// TIA Portal project "Project" (V15)

(* hardware
DEVICE "S7-1200 station_1"  S7-1200 Station
   slot 0: "Rack_0"  S7-1200 Rack  Rack  V1.0
   slot 1: "PLC_1"  CPU 1214C DC/DC/DC  6ES7 214-1AG40-0XB0  V4.2
DEVICE "HMI_1"  TP1200 Comfort
   slot 0: "HMI_1"  TP1200 Comfort  6AV2 124-0MC01-0AX0  15.0.0.0
   slot 1: "HMI_RT_1"  TP1200 Comfort  6AV2 124-0MC01-0AX0  15.0.0.0
   slot 5: "HMI_1.IE_CP_1"  PROFINET Interface  15.0.0.0
      slot 1: "PROFINET Interface_1"  PROFINET Interface
         slot 1: "Port_1"  Port
         slot 2: "Port_2"  Port
   slot 7: "HMI_1.MPI/DP_CP_1"  MPI/DP Interface  15.0.0.0
*)

// ===== PLC "PLC_1"  CPU 1214C DC/DC/DC =====

VAR_GLOBAL   // PLC tag table "Default tag table"
   "Start" AT %M0.0 : Bool;
   "Stop" AT %M0.1 : Bool;
   "Run" AT %M0.2 : Bool;
   "Low" AT %M0.3 : Bool;
   "Reset" AT %M0.4 : Bool;
   "Sensor_Low" AT %M0.5 : Bool;
   "Piston_Low" AT %Q0.0 : Bool;
   "High" AT %M0.6 : Bool;
   "Sensor_High" AT %M0.7 : Bool;
   "Piston_High" AT %Q0.1 : Bool;
   "Medium" AT %M1.0 : Bool;
   "Sensor_Medium" AT %M1.1 : Bool;
   "Piston_Medium" AT %Q0.2 : Bool;
END_VAR

DATA_BLOCK "Control_Piston_Low_DB"   // DB1
{ S7_Optimized_Access := 'TRUE' }
VERSION : 0.1
// stored: InstanceOfName Control_Piston
"Control_Piston"
BEGIN
END_DATA_BLOCK

DATA_BLOCK "Control_Piston_High_DB"   // DB2
{ S7_Optimized_Access := 'TRUE' }
VERSION : 0.1
// stored: InstanceOfName Control_Piston
"Control_Piston"
BEGIN
END_DATA_BLOCK

DATA_BLOCK "Control_Piston_Med_DB"   // DB3
{ S7_Optimized_Access := 'TRUE' }
VERSION : 0.1
// stored: InstanceOfName Control_Piston
"Control_Piston"
BEGIN
END_DATA_BLOCK

DATA_BLOCK "DB_Main"   // DB4
{ S7_Optimized_Access := 'TRUE' }
VERSION : 0.1
   VAR
      Pos_edge_1 : Bool;
      Pos_edge_2 : Bool;
      Pos_edge_3 : Bool;
      Number_of_low_boxes : Int;
      Number_of_med_boxes : Int;
      Number_of_high_boxes : Int;
   END_VAR
BEGIN
END_DATA_BLOCK

// folder: System blocks/Program resources

DATA_BLOCK "IEC_Counter_0_DB"   // DB5
{ S7_Optimized_Access := 'TRUE' }
AUTHOR : Simatic
FAMILY : IEC
NAME : CNTR
VERSION : 1.0
// stored: InstanceOfName IEC_COUNTER
"IEC_COUNTER"
BEGIN
END_DATA_BLOCK

DATA_BLOCK "IEC_Counter_1_DB"   // DB6
{ S7_Optimized_Access := 'TRUE' }
AUTHOR : Simatic
FAMILY : IEC
NAME : CNTR
VERSION : 1.0
// stored: InstanceOfName IEC_COUNTER
"IEC_COUNTER"
BEGIN
END_DATA_BLOCK

DATA_BLOCK "IEC_Counter_2_DB"   // DB7
{ S7_Optimized_Access := 'TRUE' }
AUTHOR : Simatic
FAMILY : IEC
NAME : CNTR
VERSION : 1.0
// stored: InstanceOfName IEC_COUNTER
"IEC_COUNTER"
BEGIN
END_DATA_BLOCK

// folder: (top level)

FUNCTION_BLOCK "Single_box_behaviour"   // FB1, LAD
{ S7_Optimized_Access := 'TRUE' }
VERSION : 0.1
// Khối quản lý hành vi của từng hộp
   VAR_INPUT
      Low_box_in : Bool;
      Start : Bool;
      Stop : Bool;
      Run : Bool;
      Reset : Bool;
      Maximum_time : Time;
      Maximum_time_int : Int;
   END_VAR
   VAR_OUTPUT
      Current_time : Int;
      Animation_run_out : Bool;
   END_VAR
   VAR
      Animation_run : Bool;
      IEC_Timer_0_Instance : TON_TIME;
      Low__timer_acc : Time;
      Current_time_mem : Int;
      Halting : Bool;
      Pos_edge_1 : Bool;
   END_VAR
   VAR_TEMP
      Low__timer_acc_int : Int;
   END_VAR
   VAR_TEMP   // added for the SCL form of the ladder/FBD networks
      _w1 : Bool;
   END_VAR
BEGIN

REGION Network 1
   // Cho animation chạy khi có tín hiệu xung cạnh lên hoặc tiếp tục khi đang stop
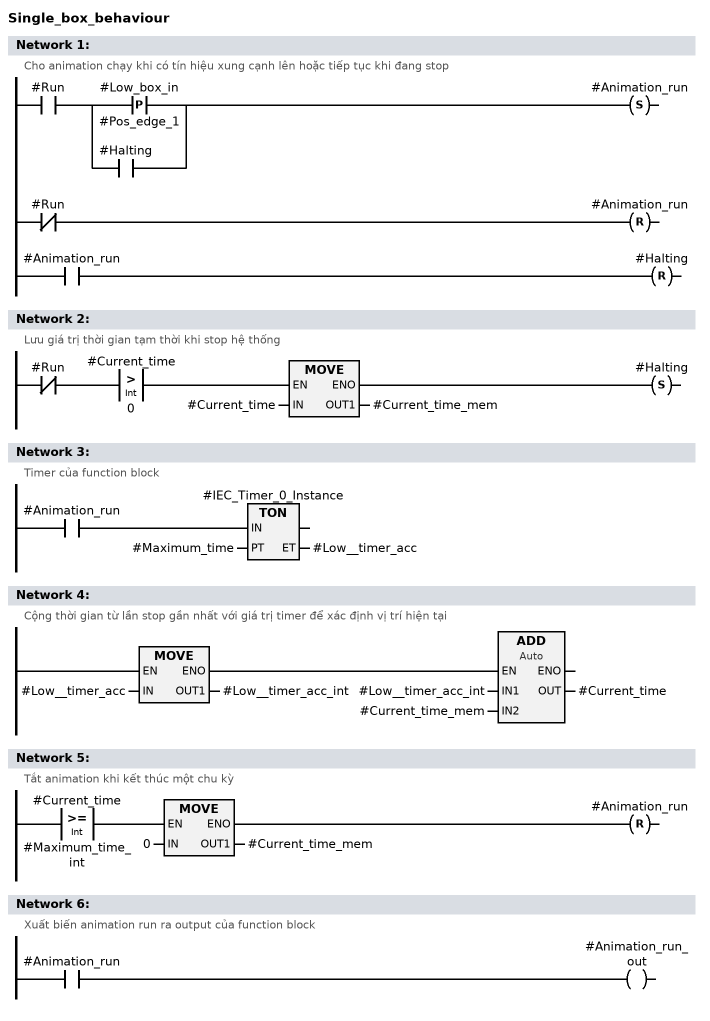
   RUNG wire#powerrail
      Contact( #Run )
      wire#w1
      P_Contact(operand := #Low_box_in, bit := #Pos_edge_1)
      wire#w2
      S_Coil( #Animation_run )
   END_RUNG
   RUNG wire#w1
      Contact( #Halting )
   END_RUNG wire#w2
   RUNG wire#powerrail
      I_Contact( #Run )
      R_Coil( #Animation_run )
   END_RUNG
   RUNG wire#powerrail
      Contact( #Animation_run )
      R_Coil( #Halting )
   END_RUNG
   // the same network as SCL:
   #_w1 := #Run AND #Low_box_in AND NOT #Pos_edge_1;   // rising edge of #Low_box_in
   #Pos_edge_1 := #Low_box_in;
   IF #_w1 OR (#Run AND #Halting) THEN #Animation_run := TRUE; END_IF;
   IF NOT #Run THEN #Animation_run := FALSE; END_IF;
   IF #Animation_run THEN #Halting := FALSE; END_IF;
END_REGION

REGION Network 2
   // Lưu giá trị thời gian tạm thời khi stop hệ thống
   RUNG wire#powerrail
      I_Contact( #Run )
      { S7_Templates := "SrcType := Int" } GT_Contact(in1 := #Current_time, in2 := 0)
      Move(in := #Current_time, out1 => #Current_time_mem)
      S_Coil( #Halting )
   END_RUNG
   // the same network as SCL:
   IF NOT #Run AND (#Current_time > 0) THEN
       #Current_time_mem := #Current_time;
       #Halting := TRUE;
   END_IF;
END_REGION

REGION Network 3
   // Timer của function block
   #IEC_Timer_0_Instance(IN := #Animation_run, PT := #Maximum_time, ET => #Low__timer_acc);   // TON
END_REGION

REGION Network 4
   // Cộng thời gian từ lần stop gần nhất với giá trị timer để xác định vị trí hiện tại
   RUNG wire#powerrail
      Move(in := #Low__timer_acc, out1 => #Low__timer_acc_int)
      Add(in1 := #Low__timer_acc_int, in2 := #Current_time_mem, out => #Current_time)
   END_RUNG
   // the same network as SCL:
   #Low__timer_acc_int := #Low__timer_acc;
   #Current_time := #Low__timer_acc_int + #Current_time_mem;
END_REGION

REGION Network 5
   // Tắt animation khi kết thúc một chu kỳ
   RUNG wire#powerrail
      { S7_Templates := "SrcType := Int" } GE_Contact(in1 := #Current_time, in2 := #Maximum_time_int)
      Move(in := 0, out1 => #Current_time_mem)
      R_Coil( #Animation_run )
   END_RUNG
   // the same network as SCL:
   IF #Current_time >= #Maximum_time_int THEN
       #Current_time_mem := 0;
       #Animation_run := FALSE;
   END_IF;
END_REGION

REGION Network 6
   // Xuất biến animation run ra output của function block
   RUNG wire#powerrail
      Contact( #Animation_run )
      Coil( #Animation_run_out )
   END_RUNG
   // the same network as SCL:
   #Animation_run_out := #Animation_run;
END_REGION
END_FUNCTION_BLOCK

FUNCTION_BLOCK "Multiple_boxes_behaviour"   // FB2, LAD
{ S7_Optimized_Access := 'TRUE' }
VERSION : 0.1
// Khối quản lý hành vi của từng nhóm hộp (thấp, trung bình, cao)
   VAR_INPUT
      Low_box_in : Bool;
      Start : Bool;
      Stop : Bool;
      Run : Bool;
      Reset : Bool;
      Maximum_time : Time;
      Maximum_time_int : Int;
      Sensor_Activate_Time : Int;
      Sensor_Deactivate_Time : Int;
   END_VAR
   VAR_OUTPUT
      Sensor : Bool;
   END_VAR
   VAR
      Neg_edge_1 : Bool;
   END_VAR
   VAR RETAIN
      IEC_Counter_0_Instance : CTUD_INT;
   END_VAR
   VAR
      Animation_1 : Bool;
      Number_of_running_graphic : Int;
      Animation_2 : Bool;
      Current_Time_1 : Int;
      Current_Time_2 : Int;
      Animation_3 : Bool;
      Load_value : Int;
      Current_Time_3 : Int;
      Count_down : Bool;
      Neg_edge_2 : Bool;
      Neg_edge_3 : Bool;
      Number_of_boxes_on_conveyor_belt : Int;
      Single_box_animation_1 : Bool;
      Single_box_animation_2 : Bool;
      Single_box_animation_3 : Bool;
      Neg_edge_4 : Bool;
      Neg_edge_5 : Bool;
      Neg_edge_6 : Bool;
      Reset_counter : Bool;
      Animation_wait : Bool;
      Pos_edge_1 : Bool;
      Single_box_animation_4 : Bool;
      Current_Time_4 : Int;
      Animation_4 : Bool;
      Neg_edge_7 : Bool;
      Single_box_animation_5 : Bool;
      Current_Time_5 : Int;
      Animation_5 : Bool;
      Neg_edge_8 : Bool;
      Neg_edge_9 : Bool;
      Neg_edge_10 : Bool;
      IEC_Timer_0_Instance : TON_TIME;
      Single_box_animation_Instance_1 : "Single_box_behaviour";
      Single_box_animation_Instance_2 : "Single_box_behaviour";
      Single_box_animation_Instance_3 : "Single_box_behaviour";
      Single_box_animation_Instance_5 : "Single_box_behaviour";
      Single_box_animation_Instance_4 : "Single_box_behaviour";
   END_VAR
   VAR_TEMP
      temp_1 : Int;
   END_VAR
   VAR_TEMP   // added for the SCL form of the ladder/FBD networks
      _w1 : Bool;
   END_VAR
BEGIN

REGION Network 1
   // Reset các animation khi có tín hiệu reset
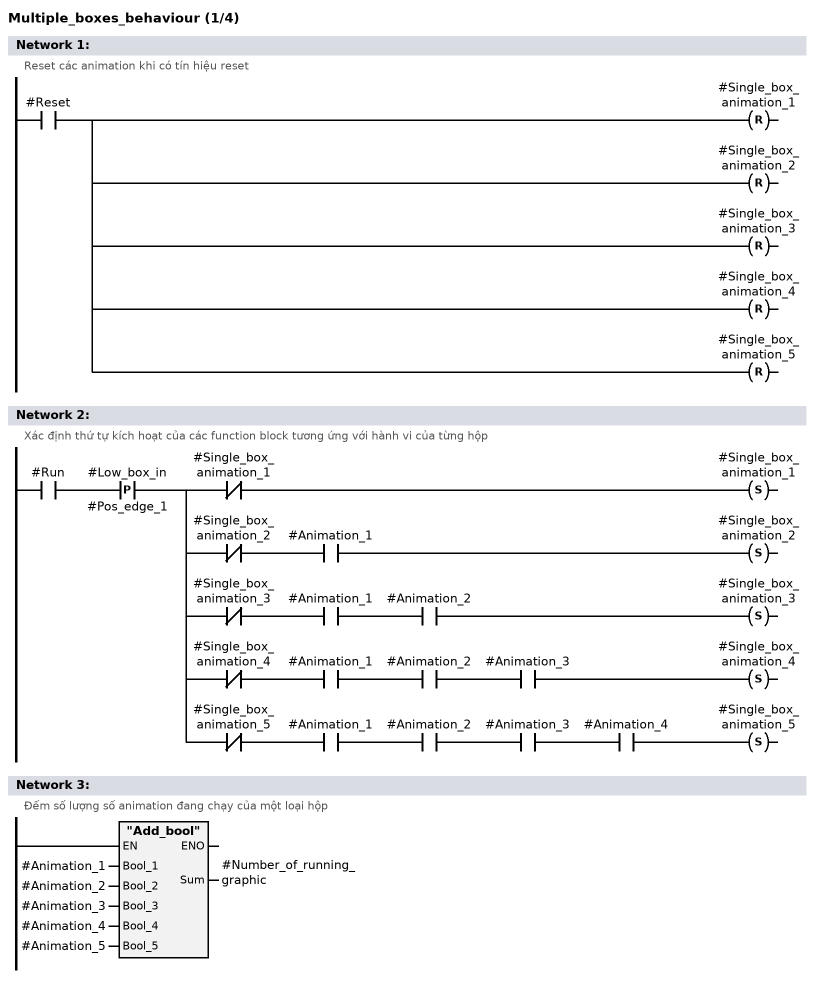
   RUNG wire#powerrail
      Contact( #Reset )
      wire#w1
      R_Coil( #Single_box_animation_1 )
   END_RUNG
   RUNG wire#w1
      R_Coil( #Single_box_animation_2 )
   END_RUNG
   RUNG wire#w1
      R_Coil( #Single_box_animation_3 )
   END_RUNG
   RUNG wire#w1
      R_Coil( #Single_box_animation_4 )
   END_RUNG
   RUNG wire#w1
      R_Coil( #Single_box_animation_5 )
   END_RUNG
   // the same network as SCL:
   IF #Reset THEN
       #Single_box_animation_1 := FALSE;
       #Single_box_animation_2 := FALSE;
       #Single_box_animation_3 := FALSE;
       #Single_box_animation_4 := FALSE;
       #Single_box_animation_5 := FALSE;
   END_IF;
END_REGION

REGION Network 2
   // Xác định thứ tự kích hoạt của các function block tương ứng với hành vi của từng hộp
   RUNG wire#powerrail
      Contact( #Run )
      P_Contact(operand := #Low_box_in, bit := #Pos_edge_1)
      wire#w1
      I_Contact( #Single_box_animation_1 )
      S_Coil( #Single_box_animation_1 )
   END_RUNG
   RUNG wire#w1
      I_Contact( #Single_box_animation_2 )
      Contact( #Animation_1 )
      S_Coil( #Single_box_animation_2 )
   END_RUNG
   RUNG wire#w1
      I_Contact( #Single_box_animation_3 )
      Contact( #Animation_1 )
      Contact( #Animation_2 )
      S_Coil( #Single_box_animation_3 )
   END_RUNG
   RUNG wire#w1
      I_Contact( #Single_box_animation_4 )
      Contact( #Animation_1 )
      Contact( #Animation_2 )
      Contact( #Animation_3 )
      S_Coil( #Single_box_animation_4 )
   END_RUNG
   RUNG wire#w1
      I_Contact( #Single_box_animation_5 )
      Contact( #Animation_1 )
      Contact( #Animation_2 )
      Contact( #Animation_3 )
      Contact( #Animation_4 )
      S_Coil( #Single_box_animation_5 )
   END_RUNG
   // the same network as SCL:
   #_w1 := #Run AND #Low_box_in AND NOT #Pos_edge_1;   // rising edge of #Low_box_in
   #Pos_edge_1 := #Low_box_in;
   IF #_w1 AND NOT #Single_box_animation_1 THEN #Single_box_animation_1 := TRUE; END_IF;
   IF #_w1 AND NOT #Single_box_animation_2 AND #Animation_1 THEN #Single_box_animation_2 := TRUE; END_IF;
   IF #_w1 AND NOT #Single_box_animation_3 AND #Animation_1 AND #Animation_2 THEN
       #Single_box_animation_3 := TRUE;
   END_IF;
   IF #_w1 AND NOT #Single_box_animation_4 AND #Animation_1 AND #Animation_2 AND #Animation_3 THEN
       #Single_box_animation_4 := TRUE;
   END_IF;
   IF #_w1 AND NOT #Single_box_animation_5 AND #Animation_1 AND #Animation_2 AND #Animation_3 AND #Animation_4 THEN
       #Single_box_animation_5 := TRUE;
   END_IF;
END_REGION

REGION Network 3
   // Đếm số lượng số animation đang chạy của một loại hộp
   RUNG wire#powerrail
      "Add_bool"(Bool_1 := #Animation_1, Bool_2 := #Animation_2, Bool_3 := #Animation_3, Bool_4 := #Animation_4, Bool_5 := #Animation_5, Sum => #Number_of_running_graphic)
   END_RUNG
   // the same network as SCL:
   "Add_bool"(Bool_1 := #Animation_1,
              Bool_2 := #Animation_2,
              Bool_3 := #Animation_3,
              Bool_4 := #Animation_4,
              Bool_5 := #Animation_5,
              Sum => #Number_of_running_graphic);
END_REGION

REGION Network 4
   // Function block xác định hành vi của hộp thứ 1
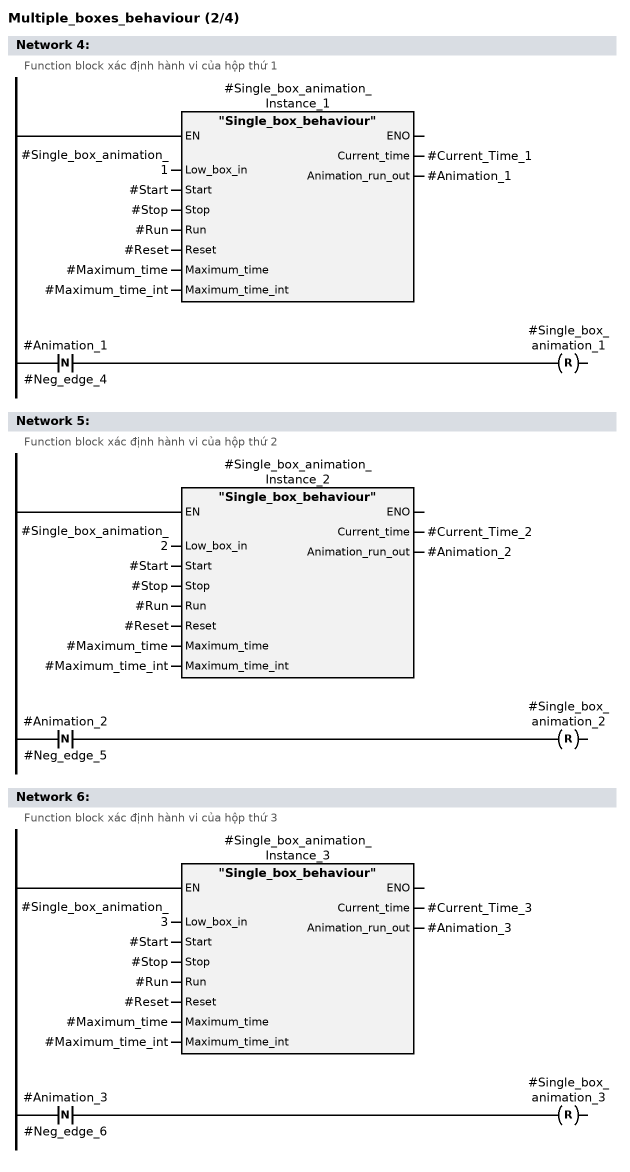
   RUNG wire#powerrail
      #Single_box_animation_Instance_1(Low_box_in := #Single_box_animation_1, Start := #Start, Stop := #Stop, Run := #Run, Reset := #Reset, Maximum_time := #Maximum_time, Maximum_time_int := #Maximum_time_int, Current_time => #Current_Time_1, Animation_run_out => #Animation_1)
   END_RUNG
   RUNG wire#powerrail
      N_Contact(operand := #Animation_1, bit := #Neg_edge_4)
      R_Coil( #Single_box_animation_1 )
   END_RUNG
   // the same network as SCL:
   #Single_box_animation_Instance_1(Low_box_in := #Single_box_animation_1,   // "Single_box_behaviour"
                           Start := #Start,
                           Stop := #Stop,
                           Run := #Run,
                           Reset := #Reset,
                           Maximum_time := #Maximum_time,
                           Maximum_time_int := #Maximum_time_int,
                           Current_time => #Current_Time_1,
                           Animation_run_out => #Animation_1);
   #_w1 := NOT #Animation_1 AND #Neg_edge_4;   // falling edge of #Animation_1
   #Neg_edge_4 := #Animation_1;
   IF #_w1 THEN #Single_box_animation_1 := FALSE; END_IF;
END_REGION

REGION Network 5
   // Function block xác định hành vi của hộp thứ 2
   RUNG wire#powerrail
      #Single_box_animation_Instance_2(Low_box_in := #Single_box_animation_2, Start := #Start, Stop := #Stop, Run := #Run, Reset := #Reset, Maximum_time := #Maximum_time, Maximum_time_int := #Maximum_time_int, Current_time => #Current_Time_2, Animation_run_out => #Animation_2)
   END_RUNG
   RUNG wire#powerrail
      N_Contact(operand := #Animation_2, bit := #Neg_edge_5)
      R_Coil( #Single_box_animation_2 )
   END_RUNG
   // the same network as SCL:
   #Single_box_animation_Instance_2(Low_box_in := #Single_box_animation_2,   // "Single_box_behaviour"
                           Start := #Start,
                           Stop := #Stop,
                           Run := #Run,
                           Reset := #Reset,
                           Maximum_time := #Maximum_time,
                           Maximum_time_int := #Maximum_time_int,
                           Current_time => #Current_Time_2,
                           Animation_run_out => #Animation_2);
   #_w1 := NOT #Animation_2 AND #Neg_edge_5;   // falling edge of #Animation_2
   #Neg_edge_5 := #Animation_2;
   IF #_w1 THEN #Single_box_animation_2 := FALSE; END_IF;
END_REGION

REGION Network 6
   // Function block xác định hành vi của hộp thứ 3
   RUNG wire#powerrail
      #Single_box_animation_Instance_3(Low_box_in := #Single_box_animation_3, Start := #Start, Stop := #Stop, Run := #Run, Reset := #Reset, Maximum_time := #Maximum_time, Maximum_time_int := #Maximum_time_int, Current_time => #Current_Time_3, Animation_run_out => #Animation_3)
   END_RUNG
   RUNG wire#powerrail
      N_Contact(operand := #Animation_3, bit := #Neg_edge_6)
      R_Coil( #Single_box_animation_3 )
   END_RUNG
   // the same network as SCL:
   #Single_box_animation_Instance_3(Low_box_in := #Single_box_animation_3,   // "Single_box_behaviour"
                           Start := #Start,
                           Stop := #Stop,
                           Run := #Run,
                           Reset := #Reset,
                           Maximum_time := #Maximum_time,
                           Maximum_time_int := #Maximum_time_int,
                           Current_time => #Current_Time_3,
                           Animation_run_out => #Animation_3);
   #_w1 := NOT #Animation_3 AND #Neg_edge_6;   // falling edge of #Animation_3
   #Neg_edge_6 := #Animation_3;
   IF #_w1 THEN #Single_box_animation_3 := FALSE; END_IF;
END_REGION

REGION Network 7
   // Function block xác định hành vi của hộp thứ 4
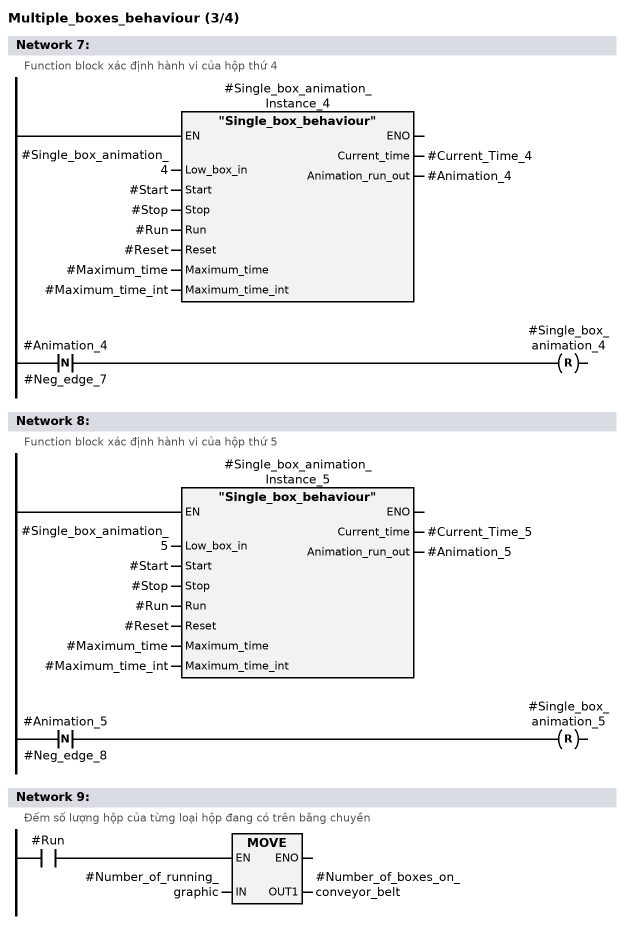
   RUNG wire#powerrail
      #Single_box_animation_Instance_4(Low_box_in := #Single_box_animation_4, Start := #Start, Stop := #Stop, Run := #Run, Reset := #Reset, Maximum_time := #Maximum_time, Maximum_time_int := #Maximum_time_int, Current_time => #Current_Time_4, Animation_run_out => #Animation_4)
   END_RUNG
   RUNG wire#powerrail
      N_Contact(operand := #Animation_4, bit := #Neg_edge_7)
      R_Coil( #Single_box_animation_4 )
   END_RUNG
   // the same network as SCL:
   #Single_box_animation_Instance_4(Low_box_in := #Single_box_animation_4,   // "Single_box_behaviour"
                           Start := #Start,
                           Stop := #Stop,
                           Run := #Run,
                           Reset := #Reset,
                           Maximum_time := #Maximum_time,
                           Maximum_time_int := #Maximum_time_int,
                           Current_time => #Current_Time_4,
                           Animation_run_out => #Animation_4);
   #_w1 := NOT #Animation_4 AND #Neg_edge_7;   // falling edge of #Animation_4
   #Neg_edge_7 := #Animation_4;
   IF #_w1 THEN #Single_box_animation_4 := FALSE; END_IF;
END_REGION

REGION Network 8
   // Function block xác định hành vi của hộp thứ 5
   RUNG wire#powerrail
      #Single_box_animation_Instance_5(Low_box_in := #Single_box_animation_5, Start := #Start, Stop := #Stop, Run := #Run, Reset := #Reset, Maximum_time := #Maximum_time, Maximum_time_int := #Maximum_time_int, Current_time => #Current_Time_5, Animation_run_out => #Animation_5)
   END_RUNG
   RUNG wire#powerrail
      N_Contact(operand := #Animation_5, bit := #Neg_edge_8)
      R_Coil( #Single_box_animation_5 )
   END_RUNG
   // the same network as SCL:
   #Single_box_animation_Instance_5(Low_box_in := #Single_box_animation_5,   // "Single_box_behaviour"
                           Start := #Start,
                           Stop := #Stop,
                           Run := #Run,
                           Reset := #Reset,
                           Maximum_time := #Maximum_time,
                           Maximum_time_int := #Maximum_time_int,
                           Current_time => #Current_Time_5,
                           Animation_run_out => #Animation_5);
   #_w1 := NOT #Animation_5 AND #Neg_edge_8;   // falling edge of #Animation_5
   #Neg_edge_8 := #Animation_5;
   IF #_w1 THEN #Single_box_animation_5 := FALSE; END_IF;
END_REGION

REGION Network 9
   // Đếm số lượng hộp của từng loại hộp đang có trên băng chuyền
   RUNG wire#powerrail
      Contact( #Run )
      Move(in := #Number_of_running_graphic, out1 => #Number_of_boxes_on_conveyor_belt)
   END_RUNG
   // the same network as SCL:
   IF #Run THEN #Number_of_boxes_on_conveyor_belt := #Number_of_running_graphic; END_IF;
END_REGION

REGION Network 10
   // Kiểm tra trạng thái của sensor dựa trên vị trí mỗi hộp
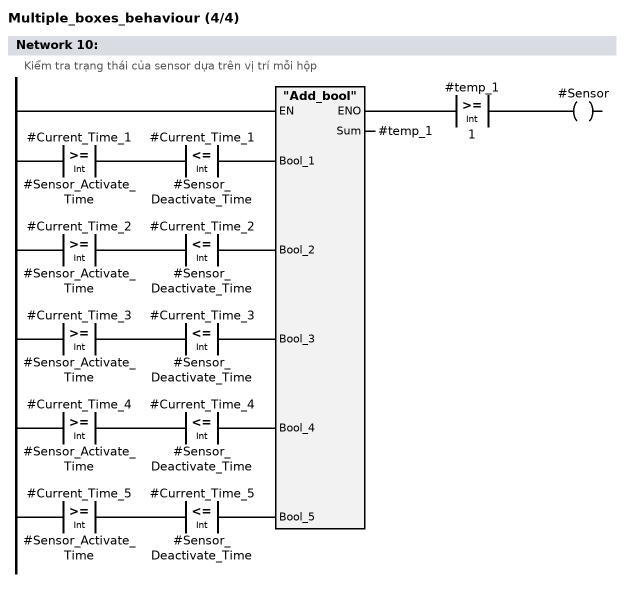
   RUNG wire#powerrail
      "Add_bool"(Bool_1 := wire#w1, Bool_2 := wire#w2, Bool_3 := wire#w3, Bool_4 := wire#w4, Bool_5 := wire#w5, Sum => #temp_1)
      { S7_Templates := "SrcType := Int" } GE_Contact(in1 := #temp_1, in2 := 1)
      Coil( #Sensor )
   END_RUNG
   RUNG wire#powerrail
      { S7_Templates := "SrcType := Int" } GE_Contact(in1 := #Current_Time_1, in2 := #Sensor_Activate_Time)
      { S7_Templates := "SrcType := Int" } LE_Contact(in1 := #Current_Time_1, in2 := #Sensor_Deactivate_Time)
   END_RUNG wire#w1
   RUNG wire#powerrail
      { S7_Templates := "SrcType := Int" } GE_Contact(in1 := #Current_Time_2, in2 := #Sensor_Activate_Time)
      { S7_Templates := "SrcType := Int" } LE_Contact(in1 := #Current_Time_2, in2 := #Sensor_Deactivate_Time)
   END_RUNG wire#w2
   RUNG wire#powerrail
      { S7_Templates := "SrcType := Int" } GE_Contact(in1 := #Current_Time_3, in2 := #Sensor_Activate_Time)
      { S7_Templates := "SrcType := Int" } LE_Contact(in1 := #Current_Time_3, in2 := #Sensor_Deactivate_Time)
   END_RUNG wire#w3
   RUNG wire#powerrail
      { S7_Templates := "SrcType := Int" } GE_Contact(in1 := #Current_Time_4, in2 := #Sensor_Activate_Time)
      { S7_Templates := "SrcType := Int" } LE_Contact(in1 := #Current_Time_4, in2 := #Sensor_Deactivate_Time)
   END_RUNG wire#w4
   RUNG wire#powerrail
      { S7_Templates := "SrcType := Int" } GE_Contact(in1 := #Current_Time_5, in2 := #Sensor_Activate_Time)
      { S7_Templates := "SrcType := Int" } LE_Contact(in1 := #Current_Time_5, in2 := #Sensor_Deactivate_Time)
   END_RUNG wire#w5
   // the same network as SCL:
   "Add_bool"(Bool_1 := (#Current_Time_1 >= #Sensor_Activate_Time) AND (#Current_Time_1 <= #Sensor_Deactivate_Time),
              Bool_2 := (#Current_Time_2 >= #Sensor_Activate_Time) AND (#Current_Time_2 <= #Sensor_Deactivate_Time),
              Bool_3 := (#Current_Time_3 >= #Sensor_Activate_Time) AND (#Current_Time_3 <= #Sensor_Deactivate_Time),
              Bool_4 := (#Current_Time_4 >= #Sensor_Activate_Time) AND (#Current_Time_4 <= #Sensor_Deactivate_Time),
              Bool_5 := (#Current_Time_5 >= #Sensor_Activate_Time) AND (#Current_Time_5 <= #Sensor_Deactivate_Time),
              Sum => #temp_1,
              ENO => #_w1);
   #Sensor := #_w1 AND (#temp_1 >= 1);
END_REGION
END_FUNCTION_BLOCK

FUNCTION_BLOCK "Control_Piston"   // FB3, LAD
{ S7_Optimized_Access := 'TRUE' }
VERSION : 0.1
// Khối xác định tín hiệu điều khiển của piston
   VAR_INPUT
      Box_in : Bool;
      Start : Bool;
      Stop : Bool;
      Run : Bool;
      Reset : Bool;
      Maximum_time : Time;
      Maximum_time_int : Int;
      Sensor_Activate_Time : Int;
      Sensor_Deactivate_Time : Int;
      Time_Interval_Sensor_To_Piston_Begin_Pushing : Time;
      Time_Interval_Sensor_To_Piston_Finish_Pushing : Time;
      Time_Interval_Sensor_To_Piston_Finish_Pushing_Int : Int;
      Time_Interval_Sensor_To_Piston_Begin_Pushing_Int : Int;
   END_VAR
   VAR_OUTPUT
      Sensor_Out : Bool;
      Piston : Bool;
   END_VAR
   VAR
      Sensor : Bool;
      IEC_Timer_0_Instance : TON_TIME;
      Pos_edge_1 : Bool;
      Timer_1_Piston : Bool;
      IEC_Timer_0_Instance_1 : TON_TIME;
      IEC_Timer_0_Instance_2 : TON_TIME;
      Timer_2_Piston : Bool;
      IEC_Timer_0_Instance_3 : TON_TIME;
      Timer_3_Piston : Bool;
      Timer_4_Piston : Bool;
      Timer_5_Piston : Bool;
      IEC_Timer_0_Instance_4 : TON_TIME;
      IEC_Timer_0_Instance_5 : TON_TIME;
      Timer_Piston_Instance_1 : "Timer_Piston";
      Timer_1_Run : Bool;
      Neg_edge_1 : Bool;
      Timer_Piston_Instance_2 : "Timer_Piston";
      Timer_2_Run : Bool;
      Timer_Piston_Instance_3 : "Timer_Piston";
      Timer_3_Run : Bool;
      Neg_edge_2 : Bool;
      Neg_edge_3 : Bool;
      Timer_Piston_Instance_4 : "Timer_Piston";
      Timer_4_Run : Bool;
      Neg_edge_4 : Bool;
      Timer_Piston_Instance_5 : "Timer_Piston";
      Timer_5_Run : Bool;
      Neg_edge_5 : Bool;
      Multiple_boxes : "Multiple_boxes_behaviour";
   END_VAR
   VAR_TEMP
      Timer_1_Value : Int;
      Timer_2_Value : Int;
      Timer_3_Value : Int;
      Timer_4_Value : Int;
      Timer_5_Value : Int;
      Sum : Int;
   END_VAR
   VAR_TEMP   // added for the SCL form of the ladder/FBD networks
      _w1 : Bool;
   END_VAR
BEGIN

REGION Network 1
   // Network xác định hành vi của nhiều hộp cùng một loại hộp
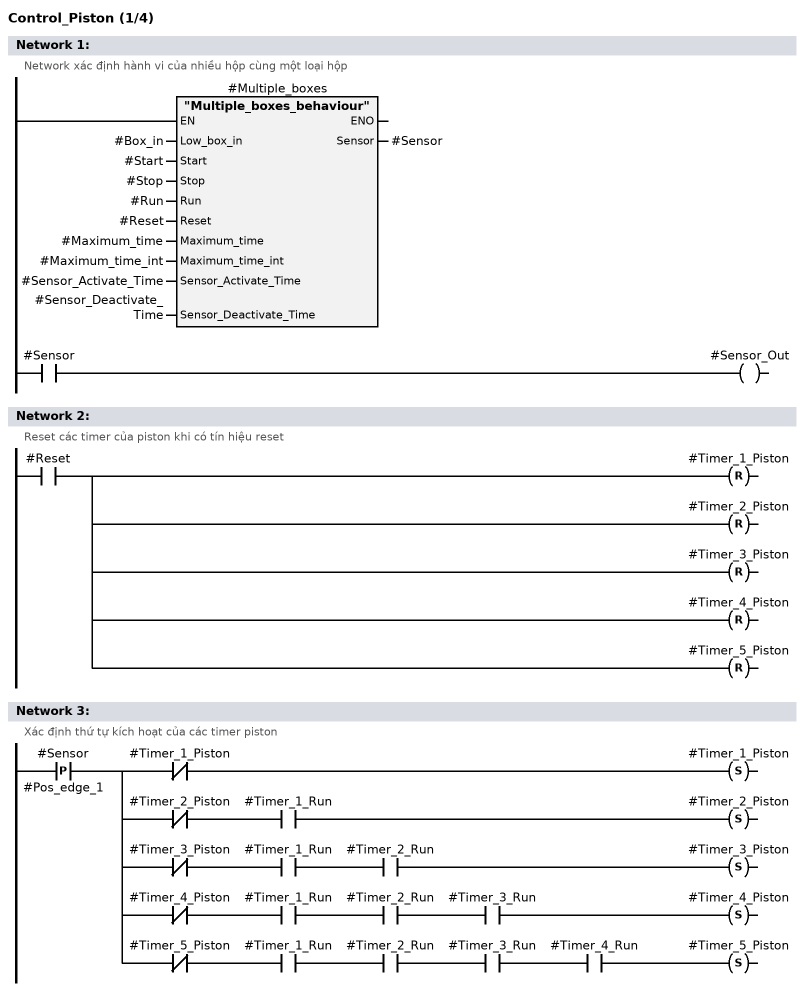
   RUNG wire#powerrail
      #Multiple_boxes(Low_box_in := #Box_in, Start := #Start, Stop := #Stop, Run := #Run, Reset := #Reset, Maximum_time := #Maximum_time, Maximum_time_int := #Maximum_time_int, Sensor_Activate_Time := #Sensor_Activate_Time, Sensor_Deactivate_Time := #Sensor_Deactivate_Time, Sensor => #Sensor)
   END_RUNG
   RUNG wire#powerrail
      Contact( #Sensor )
      Coil( #Sensor_Out )
   END_RUNG
   // the same network as SCL:
   #Multiple_boxes(Low_box_in := #Box_in,   // "Multiple_boxes_behaviour"
                   Start := #Start,
                   Stop := #Stop,
                   Run := #Run,
                   Reset := #Reset,
                   Maximum_time := #Maximum_time,
                   Maximum_time_int := #Maximum_time_int,
                   Sensor_Activate_Time := #Sensor_Activate_Time,
                   Sensor_Deactivate_Time := #Sensor_Deactivate_Time,
                   Sensor => #Sensor);
   #Sensor_Out := #Sensor;
END_REGION

REGION Network 2
   // Reset các timer của piston khi có tín hiệu reset
   RUNG wire#powerrail
      Contact( #Reset )
      wire#w1
      R_Coil( #Timer_1_Piston )
   END_RUNG
   RUNG wire#w1
      R_Coil( #Timer_2_Piston )
   END_RUNG
   RUNG wire#w1
      R_Coil( #Timer_3_Piston )
   END_RUNG
   RUNG wire#w1
      R_Coil( #Timer_4_Piston )
   END_RUNG
   RUNG wire#w1
      R_Coil( #Timer_5_Piston )
   END_RUNG
   // the same network as SCL:
   IF #Reset THEN
       #Timer_1_Piston := FALSE;
       #Timer_2_Piston := FALSE;
       #Timer_3_Piston := FALSE;
       #Timer_4_Piston := FALSE;
       #Timer_5_Piston := FALSE;
   END_IF;
END_REGION

REGION Network 3
   // Xác định thứ tự kích hoạt của các timer piston
   RUNG wire#powerrail
      P_Contact(operand := #Sensor, bit := #Pos_edge_1)
      wire#w1
      I_Contact( #Timer_1_Piston )
      S_Coil( #Timer_1_Piston )
   END_RUNG
   RUNG wire#w1
      I_Contact( #Timer_2_Piston )
      Contact( #Timer_1_Run )
      S_Coil( #Timer_2_Piston )
   END_RUNG
   RUNG wire#w1
      I_Contact( #Timer_3_Piston )
      Contact( #Timer_1_Run )
      Contact( #Timer_2_Run )
      S_Coil( #Timer_3_Piston )
   END_RUNG
   RUNG wire#w1
      I_Contact( #Timer_4_Piston )
      Contact( #Timer_1_Run )
      Contact( #Timer_2_Run )
      Contact( #Timer_3_Run )
      S_Coil( #Timer_4_Piston )
   END_RUNG
   RUNG wire#w1
      I_Contact( #Timer_5_Piston )
      Contact( #Timer_1_Run )
      Contact( #Timer_2_Run )
      Contact( #Timer_3_Run )
      Contact( #Timer_4_Run )
      S_Coil( #Timer_5_Piston )
   END_RUNG
   // the same network as SCL:
   #_w1 := #Sensor AND NOT #Pos_edge_1;   // rising edge of #Sensor
   #Pos_edge_1 := #Sensor;
   IF #_w1 AND NOT #Timer_1_Piston THEN #Timer_1_Piston := TRUE; END_IF;
   IF #_w1 AND NOT #Timer_2_Piston AND #Timer_1_Run THEN #Timer_2_Piston := TRUE; END_IF;
   IF #_w1 AND NOT #Timer_3_Piston AND #Timer_1_Run AND #Timer_2_Run THEN #Timer_3_Piston := TRUE; END_IF;
   IF #_w1 AND NOT #Timer_4_Piston AND #Timer_1_Run AND #Timer_2_Run AND #Timer_3_Run THEN
       #Timer_4_Piston := TRUE;
   END_IF;
   IF #_w1 AND NOT #Timer_5_Piston AND #Timer_1_Run AND #Timer_2_Run AND #Timer_3_Run AND #Timer_4_Run THEN
       #Timer_5_Piston := TRUE;
   END_IF;
END_REGION

REGION Network 4
   // Khối timer piston thứ 1
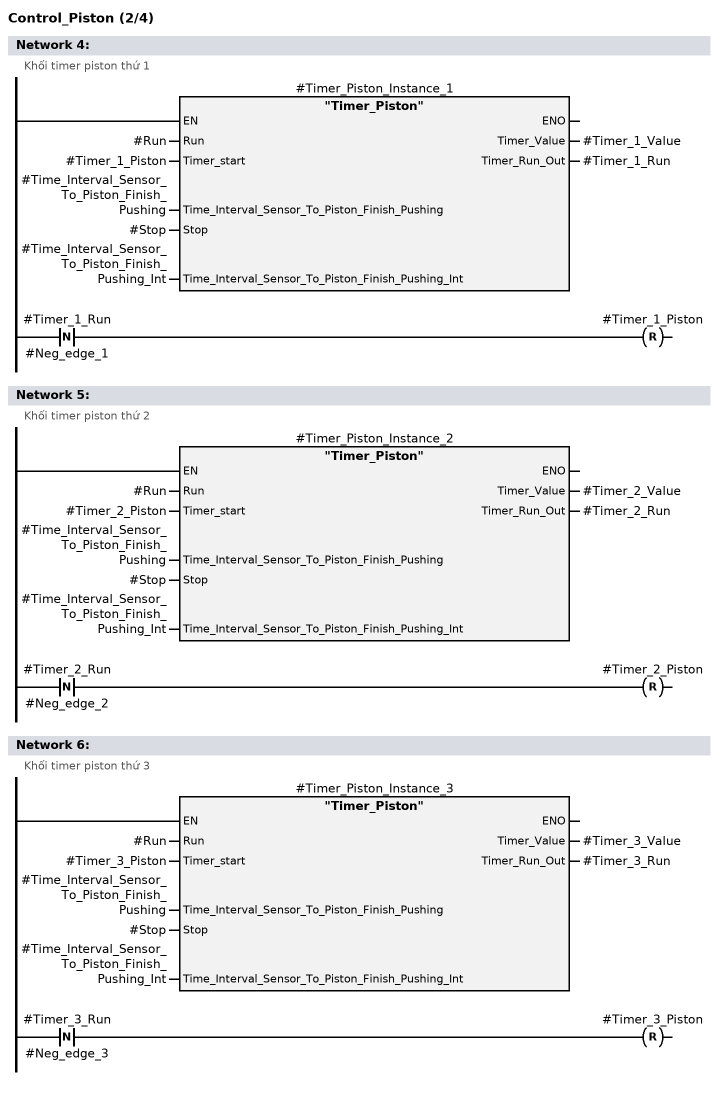
   RUNG wire#powerrail
      #Timer_Piston_Instance_1(Run := #Run, Timer_start := #Timer_1_Piston, Time_Interval_Sensor_To_Piston_Finish_Pushing := #Time_Interval_Sensor_To_Piston_Finish_Pushing, Stop := #Stop, Time_Interval_Sensor_To_Piston_Finish_Pushing_Int := #Time_Interval_Sensor_To_Piston_Finish_Pushing_Int, Timer_Value => #Timer_1_Value, Timer_Run_Out => #Timer_1_Run)
   END_RUNG
   RUNG wire#powerrail
      N_Contact(operand := #Timer_1_Run, bit := #Neg_edge_1)
      R_Coil( #Timer_1_Piston )
   END_RUNG
   // the same network as SCL:
   #Timer_Piston_Instance_1(Run := #Run,   // "Timer_Piston"
                           Timer_start := #Timer_1_Piston,
                           Time_Interval_Sensor_To_Piston_Finish_Pushing := #Time_Interval_Sensor_To_Piston_Finish_Pushing,
                           Stop := #Stop,
                           Time_Interval_Sensor_To_Piston_Finish_Pushing_Int := #Time_Interval_Sensor_To_Piston_Finish_Pushing_Int,
                           Timer_Value => #Timer_1_Value,
                           Timer_Run_Out => #Timer_1_Run);
   #_w1 := NOT #Timer_1_Run AND #Neg_edge_1;   // falling edge of #Timer_1_Run
   #Neg_edge_1 := #Timer_1_Run;
   IF #_w1 THEN #Timer_1_Piston := FALSE; END_IF;
END_REGION

REGION Network 5
   // Khối timer piston thứ 2
   RUNG wire#powerrail
      #Timer_Piston_Instance_2(Run := #Run, Timer_start := #Timer_2_Piston, Time_Interval_Sensor_To_Piston_Finish_Pushing := #Time_Interval_Sensor_To_Piston_Finish_Pushing, Stop := #Stop, Time_Interval_Sensor_To_Piston_Finish_Pushing_Int := #Time_Interval_Sensor_To_Piston_Finish_Pushing_Int, Timer_Value => #Timer_2_Value, Timer_Run_Out => #Timer_2_Run)
   END_RUNG
   RUNG wire#powerrail
      N_Contact(operand := #Timer_2_Run, bit := #Neg_edge_2)
      R_Coil( #Timer_2_Piston )
   END_RUNG
   // the same network as SCL:
   #Timer_Piston_Instance_2(Run := #Run,   // "Timer_Piston"
                           Timer_start := #Timer_2_Piston,
                           Time_Interval_Sensor_To_Piston_Finish_Pushing := #Time_Interval_Sensor_To_Piston_Finish_Pushing,
                           Stop := #Stop,
                           Time_Interval_Sensor_To_Piston_Finish_Pushing_Int := #Time_Interval_Sensor_To_Piston_Finish_Pushing_Int,
                           Timer_Value => #Timer_2_Value,
                           Timer_Run_Out => #Timer_2_Run);
   #_w1 := NOT #Timer_2_Run AND #Neg_edge_2;   // falling edge of #Timer_2_Run
   #Neg_edge_2 := #Timer_2_Run;
   IF #_w1 THEN #Timer_2_Piston := FALSE; END_IF;
END_REGION

REGION Network 6
   // Khối timer piston thứ 3
   RUNG wire#powerrail
      #Timer_Piston_Instance_3(Run := #Run, Timer_start := #Timer_3_Piston, Time_Interval_Sensor_To_Piston_Finish_Pushing := #Time_Interval_Sensor_To_Piston_Finish_Pushing, Stop := #Stop, Time_Interval_Sensor_To_Piston_Finish_Pushing_Int := #Time_Interval_Sensor_To_Piston_Finish_Pushing_Int, Timer_Value => #Timer_3_Value, Timer_Run_Out => #Timer_3_Run)
   END_RUNG
   RUNG wire#powerrail
      N_Contact(operand := #Timer_3_Run, bit := #Neg_edge_3)
      R_Coil( #Timer_3_Piston )
   END_RUNG
   // the same network as SCL:
   #Timer_Piston_Instance_3(Run := #Run,   // "Timer_Piston"
                           Timer_start := #Timer_3_Piston,
                           Time_Interval_Sensor_To_Piston_Finish_Pushing := #Time_Interval_Sensor_To_Piston_Finish_Pushing,
                           Stop := #Stop,
                           Time_Interval_Sensor_To_Piston_Finish_Pushing_Int := #Time_Interval_Sensor_To_Piston_Finish_Pushing_Int,
                           Timer_Value => #Timer_3_Value,
                           Timer_Run_Out => #Timer_3_Run);
   #_w1 := NOT #Timer_3_Run AND #Neg_edge_3;   // falling edge of #Timer_3_Run
   #Neg_edge_3 := #Timer_3_Run;
   IF #_w1 THEN #Timer_3_Piston := FALSE; END_IF;
END_REGION

REGION Network 7
   // Khối timer piston thứ 4
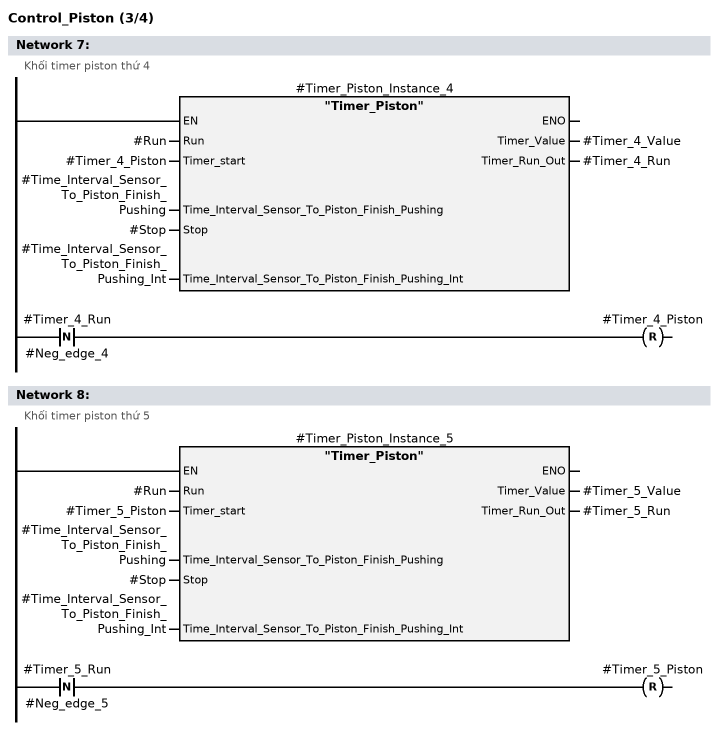
   RUNG wire#powerrail
      #Timer_Piston_Instance_4(Run := #Run, Timer_start := #Timer_4_Piston, Time_Interval_Sensor_To_Piston_Finish_Pushing := #Time_Interval_Sensor_To_Piston_Finish_Pushing, Stop := #Stop, Time_Interval_Sensor_To_Piston_Finish_Pushing_Int := #Time_Interval_Sensor_To_Piston_Finish_Pushing_Int, Timer_Value => #Timer_4_Value, Timer_Run_Out => #Timer_4_Run)
   END_RUNG
   RUNG wire#powerrail
      N_Contact(operand := #Timer_4_Run, bit := #Neg_edge_4)
      R_Coil( #Timer_4_Piston )
   END_RUNG
   // the same network as SCL:
   #Timer_Piston_Instance_4(Run := #Run,   // "Timer_Piston"
                           Timer_start := #Timer_4_Piston,
                           Time_Interval_Sensor_To_Piston_Finish_Pushing := #Time_Interval_Sensor_To_Piston_Finish_Pushing,
                           Stop := #Stop,
                           Time_Interval_Sensor_To_Piston_Finish_Pushing_Int := #Time_Interval_Sensor_To_Piston_Finish_Pushing_Int,
                           Timer_Value => #Timer_4_Value,
                           Timer_Run_Out => #Timer_4_Run);
   #_w1 := NOT #Timer_4_Run AND #Neg_edge_4;   // falling edge of #Timer_4_Run
   #Neg_edge_4 := #Timer_4_Run;
   IF #_w1 THEN #Timer_4_Piston := FALSE; END_IF;
END_REGION

REGION Network 8
   // Khối timer piston thứ 5
   RUNG wire#powerrail
      #Timer_Piston_Instance_5(Run := #Run, Timer_start := #Timer_5_Piston, Time_Interval_Sensor_To_Piston_Finish_Pushing := #Time_Interval_Sensor_To_Piston_Finish_Pushing, Stop := #Stop, Time_Interval_Sensor_To_Piston_Finish_Pushing_Int := #Time_Interval_Sensor_To_Piston_Finish_Pushing_Int, Timer_Value => #Timer_5_Value, Timer_Run_Out => #Timer_5_Run)
   END_RUNG
   RUNG wire#powerrail
      N_Contact(operand := #Timer_5_Run, bit := #Neg_edge_5)
      R_Coil( #Timer_5_Piston )
   END_RUNG
   // the same network as SCL:
   #Timer_Piston_Instance_5(Run := #Run,   // "Timer_Piston"
                           Timer_start := #Timer_5_Piston,
                           Time_Interval_Sensor_To_Piston_Finish_Pushing := #Time_Interval_Sensor_To_Piston_Finish_Pushing,
                           Stop := #Stop,
                           Time_Interval_Sensor_To_Piston_Finish_Pushing_Int := #Time_Interval_Sensor_To_Piston_Finish_Pushing_Int,
                           Timer_Value => #Timer_5_Value,
                           Timer_Run_Out => #Timer_5_Run);
   #_w1 := NOT #Timer_5_Run AND #Neg_edge_5;   // falling edge of #Timer_5_Run
   #Neg_edge_5 := #Timer_5_Run;
   IF #_w1 THEN #Timer_5_Piston := FALSE; END_IF;
END_REGION

REGION Network 9
   // Xác định trạng thái của piston
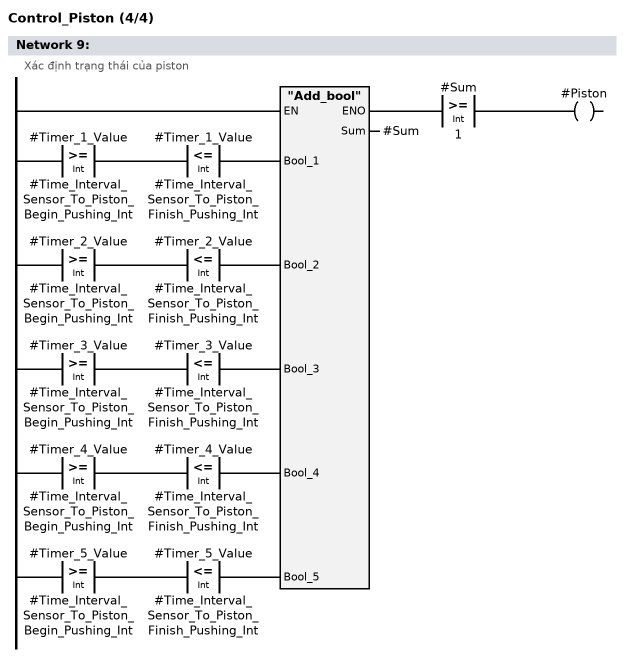
   RUNG wire#powerrail
      "Add_bool"(Bool_1 := wire#w1, Bool_2 := wire#w2, Bool_3 := wire#w3, Bool_4 := wire#w4, Bool_5 := wire#w5, Sum => #Sum)
      { S7_Templates := "SrcType := Int" } GE_Contact(in1 := #Sum, in2 := 1)
      Coil( #Piston )
   END_RUNG
   RUNG wire#powerrail
      { S7_Templates := "SrcType := Int" } GE_Contact(in1 := #Timer_1_Value, in2 := #Time_Interval_Sensor_To_Piston_Begin_Pushing_Int)
      { S7_Templates := "SrcType := Int" } LE_Contact(in1 := #Timer_1_Value, in2 := #Time_Interval_Sensor_To_Piston_Finish_Pushing_Int)
   END_RUNG wire#w1
   RUNG wire#powerrail
      { S7_Templates := "SrcType := Int" } GE_Contact(in1 := #Timer_2_Value, in2 := #Time_Interval_Sensor_To_Piston_Begin_Pushing_Int)
      { S7_Templates := "SrcType := Int" } LE_Contact(in1 := #Timer_2_Value, in2 := #Time_Interval_Sensor_To_Piston_Finish_Pushing_Int)
   END_RUNG wire#w2
   RUNG wire#powerrail
      { S7_Templates := "SrcType := Int" } GE_Contact(in1 := #Timer_3_Value, in2 := #Time_Interval_Sensor_To_Piston_Begin_Pushing_Int)
      { S7_Templates := "SrcType := Int" } LE_Contact(in1 := #Timer_3_Value, in2 := #Time_Interval_Sensor_To_Piston_Finish_Pushing_Int)
   END_RUNG wire#w3
   RUNG wire#powerrail
      { S7_Templates := "SrcType := Int" } GE_Contact(in1 := #Timer_4_Value, in2 := #Time_Interval_Sensor_To_Piston_Begin_Pushing_Int)
      { S7_Templates := "SrcType := Int" } LE_Contact(in1 := #Timer_4_Value, in2 := #Time_Interval_Sensor_To_Piston_Finish_Pushing_Int)
   END_RUNG wire#w4
   RUNG wire#powerrail
      { S7_Templates := "SrcType := Int" } GE_Contact(in1 := #Timer_5_Value, in2 := #Time_Interval_Sensor_To_Piston_Begin_Pushing_Int)
      { S7_Templates := "SrcType := Int" } LE_Contact(in1 := #Timer_5_Value, in2 := #Time_Interval_Sensor_To_Piston_Finish_Pushing_Int)
   END_RUNG wire#w5
   // the same network as SCL:
   "Add_bool"(Bool_1 := (#Timer_1_Value >= #Time_Interval_Sensor_To_Piston_Begin_Pushing_Int) AND (#Timer_1_Value <= #Time_Interval_Sensor_To_Piston_Finish_Pushing_Int),
              Bool_2 := (#Timer_2_Value >= #Time_Interval_Sensor_To_Piston_Begin_Pushing_Int) AND (#Timer_2_Value <= #Time_Interval_Sensor_To_Piston_Finish_Pushing_Int),
              Bool_3 := (#Timer_3_Value >= #Time_Interval_Sensor_To_Piston_Begin_Pushing_Int) AND (#Timer_3_Value <= #Time_Interval_Sensor_To_Piston_Finish_Pushing_Int),
              Bool_4 := (#Timer_4_Value >= #Time_Interval_Sensor_To_Piston_Begin_Pushing_Int) AND (#Timer_4_Value <= #Time_Interval_Sensor_To_Piston_Finish_Pushing_Int),
              Bool_5 := (#Timer_5_Value >= #Time_Interval_Sensor_To_Piston_Begin_Pushing_Int) AND (#Timer_5_Value <= #Time_Interval_Sensor_To_Piston_Finish_Pushing_Int),
              Sum => #Sum,
              ENO => #_w1);
   #Piston := #_w1 AND (#Sum >= 1);
END_REGION
END_FUNCTION_BLOCK

FUNCTION_BLOCK "Timer_Piston"   // FB4, LAD
{ S7_Optimized_Access := 'TRUE' }
VERSION : 0.1
// Timer của piston
   VAR_INPUT
      Run : Bool;
      Timer_start : Bool;
      Time_Interval_Sensor_To_Piston_Finish_Pushing : Time;
      Stop : Bool;
      Time_Interval_Sensor_To_Piston_Finish_Pushing_Int : Int;
   END_VAR
   VAR_OUTPUT
      Timer_Value : Int;
      Timer_Run_Out : Bool;
   END_VAR
   VAR
      Timer_Value_mem : Int;
      Halting : Bool;
      Timer_0 : TON_TIME;
      Timer_value_acc : Time;
      Pos_edge_1 : Bool;
      Timer_Run : Bool;
      IEC_Timer_0_Instance : TON_TIME;
   END_VAR
   VAR_TEMP
      Timer_value_acc_int : Int;
   END_VAR
   VAR_TEMP   // added for the SCL form of the ladder/FBD networks
      _w1 : Bool;
   END_VAR
BEGIN

REGION Network 1
   // Cho timer chạy khi có tín hiệu xung cạnh lên từ cảm biến hoặc tiếp tục khi đang stop
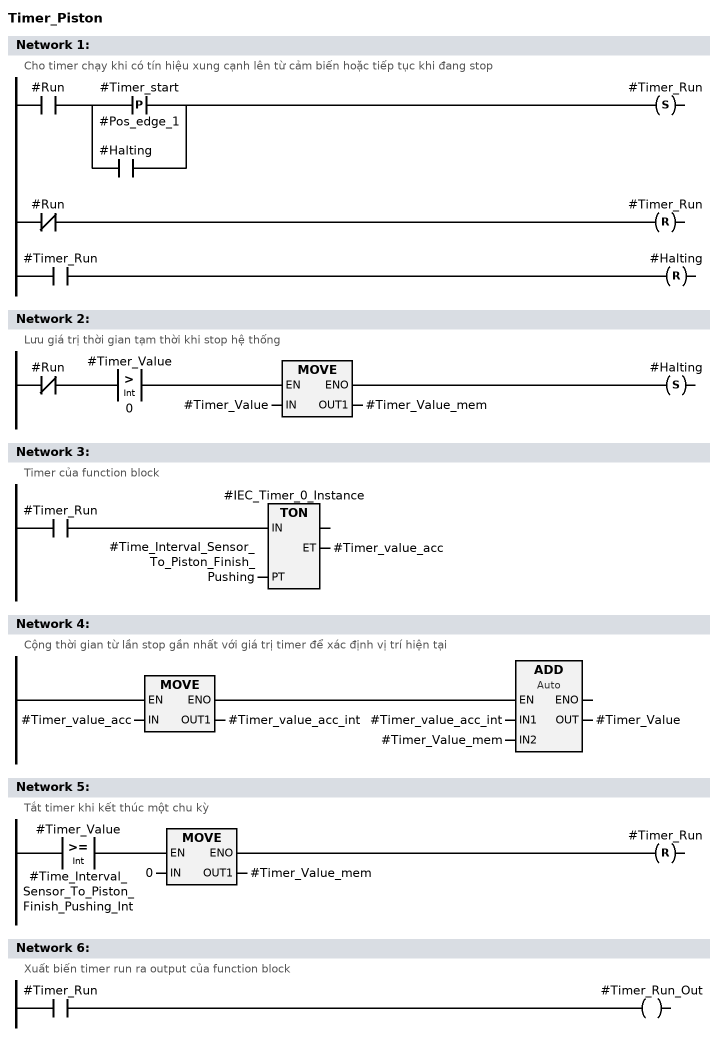
   RUNG wire#powerrail
      Contact( #Run )
      wire#w1
      P_Contact(operand := #Timer_start, bit := #Pos_edge_1)
      wire#w2
      S_Coil( #Timer_Run )
   END_RUNG
   RUNG wire#w1
      Contact( #Halting )
   END_RUNG wire#w2
   RUNG wire#powerrail
      I_Contact( #Run )
      R_Coil( #Timer_Run )
   END_RUNG
   RUNG wire#powerrail
      Contact( #Timer_Run )
      R_Coil( #Halting )
   END_RUNG
   // the same network as SCL:
   #_w1 := #Run AND #Timer_start AND NOT #Pos_edge_1;   // rising edge of #Timer_start
   #Pos_edge_1 := #Timer_start;
   IF #_w1 OR (#Run AND #Halting) THEN #Timer_Run := TRUE; END_IF;
   IF NOT #Run THEN #Timer_Run := FALSE; END_IF;
   IF #Timer_Run THEN #Halting := FALSE; END_IF;
END_REGION

REGION Network 2
   // Lưu giá trị thời gian tạm thời khi stop hệ thống
   RUNG wire#powerrail
      I_Contact( #Run )
      { S7_Templates := "SrcType := Int" } GT_Contact(in1 := #Timer_Value, in2 := 0)
      Move(in := #Timer_Value, out1 => #Timer_Value_mem)
      S_Coil( #Halting )
   END_RUNG
   // the same network as SCL:
   IF NOT #Run AND (#Timer_Value > 0) THEN
       #Timer_Value_mem := #Timer_Value;
       #Halting := TRUE;
   END_IF;
END_REGION

REGION Network 3
   // Timer của function block
   #IEC_Timer_0_Instance(IN := #Timer_Run,   // TON
                         PT := #Time_Interval_Sensor_To_Piston_Finish_Pushing,
                         ET => #Timer_value_acc);
END_REGION

REGION Network 4
   // Cộng thời gian từ lần stop gần nhất với giá trị timer để xác định vị trí hiện tại
   RUNG wire#powerrail
      Move(in := #Timer_value_acc, out1 => #Timer_value_acc_int)
      Add(in1 := #Timer_value_acc_int, in2 := #Timer_Value_mem, out => #Timer_Value)
   END_RUNG
   // the same network as SCL:
   #Timer_value_acc_int := #Timer_value_acc;
   #Timer_Value := #Timer_value_acc_int + #Timer_Value_mem;
END_REGION

REGION Network 5
   // Tắt timer khi kết thúc một chu kỳ
   RUNG wire#powerrail
      { S7_Templates := "SrcType := Int" } GE_Contact(in1 := #Timer_Value, in2 := #Time_Interval_Sensor_To_Piston_Finish_Pushing_Int)
      Move(in := 0, out1 => #Timer_Value_mem)
      R_Coil( #Timer_Run )
   END_RUNG
   // the same network as SCL:
   IF #Timer_Value >= #Time_Interval_Sensor_To_Piston_Finish_Pushing_Int THEN
       #Timer_Value_mem := 0;
       #Timer_Run := FALSE;
   END_IF;
END_REGION

REGION Network 6
   // Xuất biến timer run ra output của function block
   RUNG wire#powerrail
      Contact( #Timer_Run )
      Coil( #Timer_Run_Out )
   END_RUNG
   // the same network as SCL:
   #Timer_Run_Out := #Timer_Run;
END_REGION
END_FUNCTION_BLOCK

FUNCTION "Add_bool" : Void   // FC1, LAD
{ S7_Optimized_Access := 'TRUE' }
VERSION : 0.1
// Kiểm tra có bao nhiêu giá trị bool có giá trị 1
   VAR_INPUT
      Bool_1 : Bool;
      Bool_2 : Bool;
      Bool_3 : Bool;
      Bool_4 : Bool;
      Bool_5 : Bool;
   END_VAR
   VAR_OUTPUT
      Sum : Int;
   END_VAR
   VAR_TEMP
      temp_1 : Int;
      temp_2 : Int;
      temp_3 : Int;
      temp_4 : Int;
      temp_5 : Int;
   END_VAR
BEGIN

REGION Network 1
   // Chuyển từ giá trị bool sang int
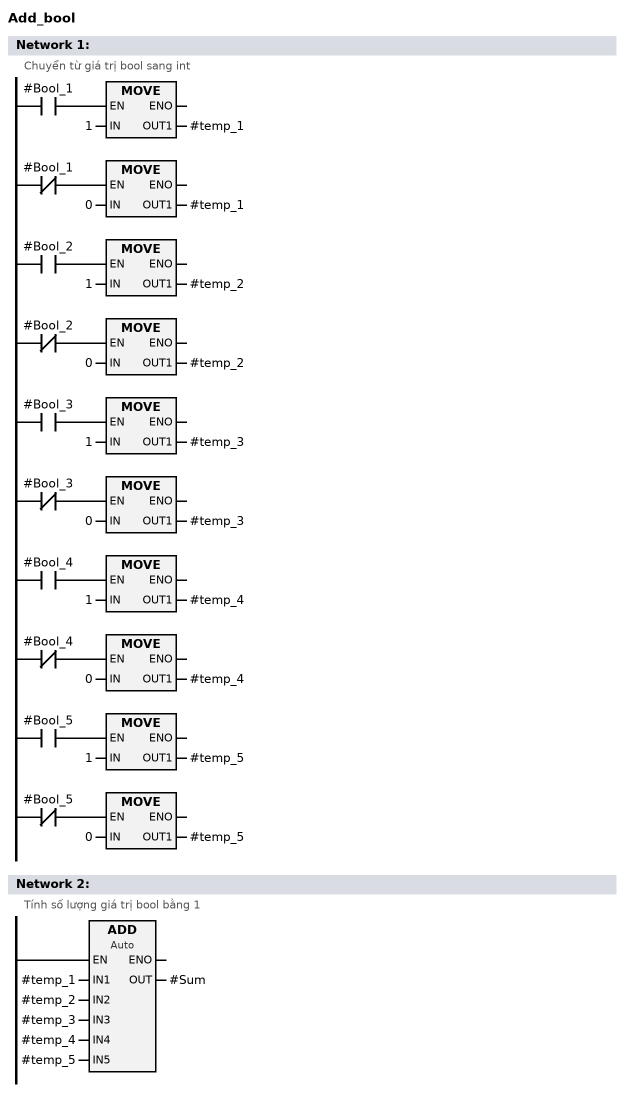
   RUNG wire#powerrail
      Contact( #Bool_1 )
      Move(in := 1, out1 => #temp_1)
   END_RUNG
   RUNG wire#powerrail
      I_Contact( #Bool_1 )
      Move(in := 0, out1 => #temp_1)
   END_RUNG
   RUNG wire#powerrail
      Contact( #Bool_2 )
      Move(in := 1, out1 => #temp_2)
   END_RUNG
   RUNG wire#powerrail
      I_Contact( #Bool_2 )
      Move(in := 0, out1 => #temp_2)
   END_RUNG
   RUNG wire#powerrail
      Contact( #Bool_3 )
      Move(in := 1, out1 => #temp_3)
   END_RUNG
   RUNG wire#powerrail
      I_Contact( #Bool_3 )
      Move(in := 0, out1 => #temp_3)
   END_RUNG
   RUNG wire#powerrail
      Contact( #Bool_4 )
      Move(in := 1, out1 => #temp_4)
   END_RUNG
   RUNG wire#powerrail
      I_Contact( #Bool_4 )
      Move(in := 0, out1 => #temp_4)
   END_RUNG
   RUNG wire#powerrail
      Contact( #Bool_5 )
      Move(in := 1, out1 => #temp_5)
   END_RUNG
   RUNG wire#powerrail
      I_Contact( #Bool_5 )
      Move(in := 0, out1 => #temp_5)
   END_RUNG
   // the same network as SCL:
   IF #Bool_1 THEN #temp_1 := 1; END_IF;
   IF NOT #Bool_1 THEN #temp_1 := 0; END_IF;
   IF #Bool_2 THEN #temp_2 := 1; END_IF;
   IF NOT #Bool_2 THEN #temp_2 := 0; END_IF;
   IF #Bool_3 THEN #temp_3 := 1; END_IF;
   IF NOT #Bool_3 THEN #temp_3 := 0; END_IF;
   IF #Bool_4 THEN #temp_4 := 1; END_IF;
   IF NOT #Bool_4 THEN #temp_4 := 0; END_IF;
   IF #Bool_5 THEN #temp_5 := 1; END_IF;
   IF NOT #Bool_5 THEN #temp_5 := 0; END_IF;
END_REGION

REGION Network 2
   // Tính số lượng giá trị bool bằng 1
   RUNG wire#powerrail
      Add(in1 := #temp_1, in2 := #temp_2, in3 := #temp_3, in4 := #temp_4, in5 := #temp_5, out => #Sum)
   END_RUNG
   // the same network as SCL:
   #Sum := #temp_1 + #temp_2 + #temp_3 + #temp_4 + #temp_5;
END_REGION
END_FUNCTION

ORGANIZATION_BLOCK "Main"   // OB1, LAD, ProgramCycle
TITLE = "Main Program Sweep (Cycle)"
{ S7_Optimized_Access := 'TRUE' }
VERSION : 0.1
// Chương trình chạy animation và xác định hoạt động của hệ thống
   VAR_INPUT
      Initial_Call : Bool;   // Initial call of this OB
      Remanence : Bool;   // =True, if remanent data are available
   END_VAR
BEGIN

REGION Network 1
   // Xác định trạng thái biến run
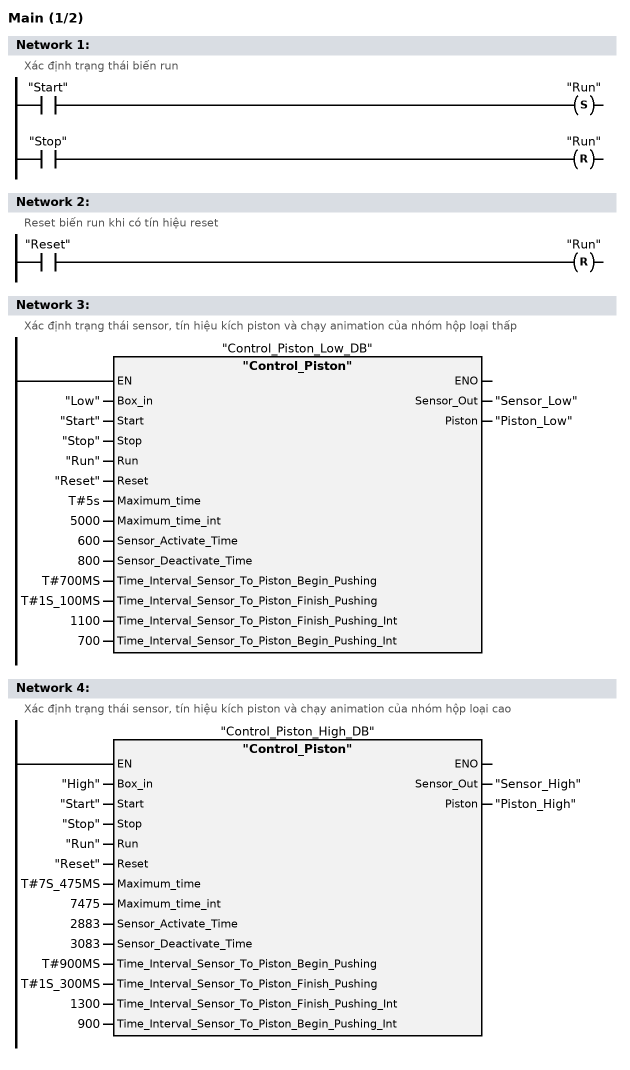
   RUNG wire#powerrail
      Contact( "Start" )
      S_Coil( "Run" )
   END_RUNG
   RUNG wire#powerrail
      Contact( "Stop" )
      R_Coil( "Run" )
   END_RUNG
   // the same network as SCL:
   IF "Start" THEN "Run" := TRUE; END_IF;
   IF "Stop" THEN "Run" := FALSE; END_IF;
END_REGION

REGION Network 2
   // Reset biến run khi có tín hiệu reset
   RUNG wire#powerrail
      Contact( "Reset" )
      R_Coil( "Run" )
   END_RUNG
   // the same network as SCL:
   IF "Reset" THEN "Run" := FALSE; END_IF;
END_REGION

REGION Network 3
   // Xác định trạng thái sensor, tín hiệu kích piston và chạy animation của nhóm hộp loại thấp
   RUNG wire#powerrail
      "Control_Piston_Low_DB"(Box_in := "Low", Start := "Start", Stop := "Stop", Run := "Run", Reset := "Reset", Maximum_time := T#5s, Maximum_time_int := 5000, Sensor_Activate_Time := 600, Sensor_Deactivate_Time := 800, Time_Interval_Sensor_To_Piston_Begin_Pushing := T#700MS, Time_Interval_Sensor_To_Piston_Finish_Pushing := T#1S_100MS, Time_Interval_Sensor_To_Piston_Finish_Pushing_Int := 1100, Time_Interval_Sensor_To_Piston_Begin_Pushing_Int := 700, Sensor_Out => "Sensor_Low", Piston => "Piston_Low")
   END_RUNG
   // the same network as SCL:
   "Control_Piston_Low_DB"(Box_in := "Low",   // "Control_Piston"
                           Start := "Start",
                           Stop := "Stop",
                           Run := "Run",
                           Reset := "Reset",
                           Maximum_time := T#5s,
                           Maximum_time_int := 5000,
                           Sensor_Activate_Time := 600,
                           Sensor_Deactivate_Time := 800,
                           Time_Interval_Sensor_To_Piston_Begin_Pushing := T#700MS,
                           Time_Interval_Sensor_To_Piston_Finish_Pushing := T#1S_100MS,
                           Time_Interval_Sensor_To_Piston_Finish_Pushing_Int := 1100,
                           Time_Interval_Sensor_To_Piston_Begin_Pushing_Int := 700,
                           Sensor_Out => "Sensor_Low",
                           Piston => "Piston_Low");
END_REGION

REGION Network 4
   // Xác định trạng thái sensor, tín hiệu kích piston và chạy animation của nhóm hộp loại cao
   RUNG wire#powerrail
      "Control_Piston_High_DB"(Box_in := "High", Start := "Start", Stop := "Stop", Run := "Run", Reset := "Reset", Maximum_time := T#7S_475MS, Maximum_time_int := 7475, Sensor_Activate_Time := 2883, Sensor_Deactivate_Time := 3083, Time_Interval_Sensor_To_Piston_Begin_Pushing := T#900MS, Time_Interval_Sensor_To_Piston_Finish_Pushing := T#1S_300MS, Time_Interval_Sensor_To_Piston_Finish_Pushing_Int := 1300, Time_Interval_Sensor_To_Piston_Begin_Pushing_Int := 900, Sensor_Out => "Sensor_High", Piston => "Piston_High")
   END_RUNG
   // the same network as SCL:
   "Control_Piston_High_DB"(Box_in := "High",   // "Control_Piston"
                           Start := "Start",
                           Stop := "Stop",
                           Run := "Run",
                           Reset := "Reset",
                           Maximum_time := T#7S_475MS,
                           Maximum_time_int := 7475,
                           Sensor_Activate_Time := 2883,
                           Sensor_Deactivate_Time := 3083,
                           Time_Interval_Sensor_To_Piston_Begin_Pushing := T#900MS,
                           Time_Interval_Sensor_To_Piston_Finish_Pushing := T#1S_300MS,
                           Time_Interval_Sensor_To_Piston_Finish_Pushing_Int := 1300,
                           Time_Interval_Sensor_To_Piston_Begin_Pushing_Int := 900,
                           Sensor_Out => "Sensor_High",
                           Piston => "Piston_High");
END_REGION

REGION Network 5
   // Xác định trạng thái sensor, tín hiệu kích piston và chạy animation của nhóm hộp loại trung bình
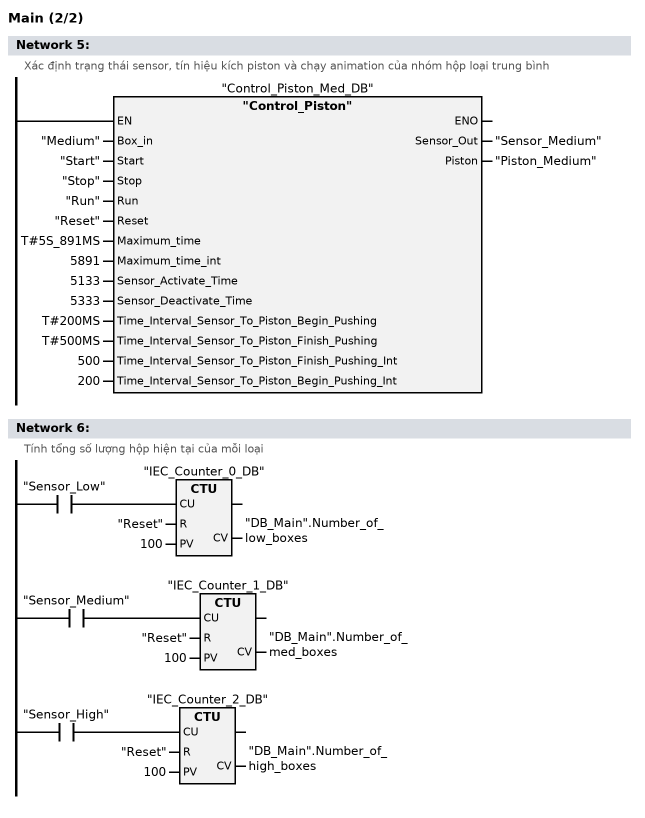
   RUNG wire#powerrail
      "Control_Piston_Med_DB"(Box_in := "Medium", Start := "Start", Stop := "Stop", Run := "Run", Reset := "Reset", Maximum_time := T#5S_891MS, Maximum_time_int := 5891, Sensor_Activate_Time := 5133, Sensor_Deactivate_Time := 5333, Time_Interval_Sensor_To_Piston_Begin_Pushing := T#200MS, Time_Interval_Sensor_To_Piston_Finish_Pushing := T#500MS, Time_Interval_Sensor_To_Piston_Finish_Pushing_Int := 500, Time_Interval_Sensor_To_Piston_Begin_Pushing_Int := 200, Sensor_Out => "Sensor_Medium", Piston => "Piston_Medium")
   END_RUNG
   // the same network as SCL:
   "Control_Piston_Med_DB"(Box_in := "Medium",   // "Control_Piston"
                           Start := "Start",
                           Stop := "Stop",
                           Run := "Run",
                           Reset := "Reset",
                           Maximum_time := T#5S_891MS,
                           Maximum_time_int := 5891,
                           Sensor_Activate_Time := 5133,
                           Sensor_Deactivate_Time := 5333,
                           Time_Interval_Sensor_To_Piston_Begin_Pushing := T#200MS,
                           Time_Interval_Sensor_To_Piston_Finish_Pushing := T#500MS,
                           Time_Interval_Sensor_To_Piston_Finish_Pushing_Int := 500,
                           Time_Interval_Sensor_To_Piston_Begin_Pushing_Int := 200,
                           Sensor_Out => "Sensor_Medium",
                           Piston => "Piston_Medium");
END_REGION

REGION Network 6
   // Tính tổng số lượng hộp hiện tại của mỗi loại
   "IEC_Counter_0_DB".CTU(CU := "Sensor_Low", R := "Reset", PV := 100, CV => "DB_Main".Number_of_low_boxes);
   "IEC_Counter_1_DB".CTU(CU := "Sensor_Medium", R := "Reset", PV := 100, CV => "DB_Main".Number_of_med_boxes);
   "IEC_Counter_2_DB".CTU(CU := "Sensor_High", R := "Reset", PV := 100, CV => "DB_Main".Number_of_high_boxes);
END_REGION
END_ORGANIZATION_BLOCK

(* ===== HMI "HMI_RT_1" =====
system functions are stored by id; their names below are inferred from use
connection "HMI_Connection_1": ETHERNET, S7_1200_OMS

HMI tags "Default tag table"
   "Start" : Bool = PLC Start AT %M0.0, 100 ms
   "Stop" : Bool = PLC Stop AT %M0.1, 100 ms
   "Low" : Bool = PLC Low AT %M0.3, 100 ms
   "Low_box_DB_Current_Time_1" : Int = PLC Control_Piston_Low_DB.Multiple_boxes.Current_Time_1, 100 ms
   "Low_box_DB_Current_Time_2" : Int = PLC Control_Piston_Low_DB.Multiple_boxes.Current_Time_2, 100 ms
   "Low_box_DB_Current_Time_3" : Int = PLC Control_Piston_Low_DB.Multiple_boxes.Current_Time_3, 100 ms
   "Reset" : Bool = PLC Reset AT %M0.4, 100 ms
   "Low_box_DB_Current_Time_4" : Int = PLC Control_Piston_Low_DB.Multiple_boxes.Current_Time_4, 100 ms
   "Low_box_DB_Current_Time_5" : Int = PLC Control_Piston_Low_DB.Multiple_boxes.Current_Time_5, 100 ms
   "Low_box_DB_Number_of_boxes_on_conveyor_belt" : Int = PLC Control_Piston_Low_DB.Multiple_boxes.Current_Time_5, 100 ms
   "Sensor_Low" : Bool = PLC Sensor_Low AT %M0.5, 100 ms
   "Piston_Low" : Bool = PLC Piston_Low AT %Q0.0, 100 ms
   "Control_Piston_Low_DB_Multiple_boxes_Number_of_boxes_on_conveyor_belt" : Int = PLC Control_Piston_Low_DB.Multiple_boxes.Number_of_boxes_on_conveyor_belt, 100 ms
   "Run" : Bool = PLC Run AT %M0.2, 100 ms
   "Control_Piston_High_DB_Multiple_boxes_Current_Time_1" : Int = PLC Control_Piston_High_DB.Multiple_boxes.Current_Time_1, 100 ms
   "Sensor_High" : Bool = PLC Sensor_High AT %M0.7, 100 ms
   "Piston_High" : Bool = PLC Piston_High AT %Q0.1, 100 ms
   "High" : Bool = PLC High AT %M0.6, 100 ms
   "Control_Piston_High_DB_Multiple_boxes_Current_Time_2" : Int = PLC Control_Piston_High_DB.Multiple_boxes.Current_Time_2, 100 ms
   "Control_Piston_High_DB_Multiple_boxes_Current_Time_3" : Int = PLC Control_Piston_High_DB.Multiple_boxes.Current_Time_3, 100 ms
   "Control_Piston_High_DB_Multiple_boxes_Current_Time_4" : Int = PLC Control_Piston_High_DB.Multiple_boxes.Current_Time_4, 100 ms
   "Control_Piston_High_DB_Multiple_boxes_Current_Time_5" : Int = PLC Control_Piston_High_DB.Multiple_boxes.Current_Time_5, 100 ms
   "Control_Piston_Med_DB_Multiple_boxes_Current_Time_1" : Int = PLC Control_Piston_Med_DB.Multiple_boxes.Current_Time_1, 100 ms
   "Control_Piston_Med_DB_Multiple_boxes_Current_Time_2" : Int = PLC Control_Piston_Med_DB.Multiple_boxes.Current_Time_2, 100 ms
   "Control_Piston_Med_DB_Multiple_boxes_Current_Time_3" : Int = PLC Control_Piston_Med_DB.Multiple_boxes.Current_Time_3, 100 ms
   "Control_Piston_Med_DB_Multiple_boxes_Current_Time_4" : Int = PLC Control_Piston_Med_DB.Multiple_boxes.Current_Time_4, 100 ms
   "Control_Piston_Med_DB_Multiple_boxes_Current_Time_5" : Int = PLC Control_Piston_Med_DB.Multiple_boxes.Current_Time_5, 100 ms
   "Medium" : Bool = PLC Medium AT %M1.0, 100 ms
   "DB_Main_Number_of_low_boxes" : Int = PLC DB_Main.Number_of_low_boxes, 100 ms
   "DB_Main_Number_of_med_boxes" : Int = PLC DB_Main.Number_of_med_boxes, 100 ms
   "DB_Main_Number_of_high_boxes" : Int = PLC DB_Main.Number_of_high_boxes, 100 ms
   "Sensor_Medium" : Bool = PLC Sensor_Medium AT %M1.1, 100 ms

screen "Screen_1" 1280x800
   GraphicView "Graphic view_3" at 367,109 size 56x134; Picture "Graphic_18"
   Button "Button_1" at 26,110 size 85x50; TextOff 'Start'
      on Press: SetBit("Start")
      on Release: ResetBit("Start")
   GraphicView "Graphic view_2" at 132,361 size 92x66; Picture "Graphic_27"
   GraphicView "Graphic view_7" at 681,105 size 56x134; Picture "Graphic_18"
   GraphicView "Graphic view_9" at 1124,16 size 80x49; Picture "Graphic_30"
   GraphicView "Graphic view_15" at 507,240 size 71x78; Picture "Graphic_44"
   GraphicView "Graphic view_1" at 249,312 size 801x60; Picture "Graphic_2"
   GraphicView "Graphic view_11" at 231,339 size 273x160; Picture "Graphic_28"
   Button "Button_2" at 27,182 size 85x50; TextOff 'Stop'
      on Release: ResetBit("Stop")
      on Press: SetBit("Stop")
   Button "Button_3" at 140,182 size 85x50; TextOff 'High'
      on Press: SetBit("High")
      on Release: ResetBit("High")
   GraphicView "Graphic view_4" at 520,339 size 273x160; Picture "Graphic_28"
   Button "Button_4" at 27,46 size 85x50; TextOff 'Reset'
      on Release: ResetBit("Reset")
      on Press: SetBit("Reset")
   IOField "I/O field_1" at 443,73 size 61x36; FormatPattern 999
      ProcessValue <- "DB_Main_Number_of_low_boxes"
   Circle "Circle_1" at 376,64 size 36x36
      Appearance <- "Sensor_Low"
   GraphicView "Graphic view_26" at 492,274 size 57x56; Picture "Graphic_55"
      Visibility <- "Piston_Low"
   Circle "Circle_2" at 528,203 size 28x28
      Appearance <- "Piston_Low"
   GraphicView "Graphic view_5" at 464,301 size 64x38; Picture "Graphic_25"
      DiagonalMovement <- "Low_box_DB_Current_Time_1"
      Visibility <- "Low_box_DB_Current_Time_1"
   GraphicView "Graphic view_13" at 464,301 size 64x38; Picture "Graphic_25"
      DiagonalMovement <- "Low_box_DB_Current_Time_2"
      Visibility <- "Low_box_DB_Current_Time_2"
   GraphicView "Graphic view_6" at 464,301 size 64x38; Picture "Graphic_25"
      DiagonalMovement <- "Low_box_DB_Current_Time_3"
      Visibility <- "Low_box_DB_Current_Time_3"
   GraphicView "Graphic view_14" at 464,301 size 64x38; Picture "Graphic_25"
      DiagonalMovement <- "Low_box_DB_Current_Time_4"
      Visibility <- "Low_box_DB_Current_Time_4"
   GraphicView "Graphic view_16" at 464,301 size 64x38; Picture "Graphic_25"
      DiagonalMovement <- "Low_box_DB_Current_Time_5"
      Visibility <- "Low_box_DB_Current_Time_5"
   GraphicView "Graphic view_17" at 283,301 size 64x38; Picture "Graphic_25"
      Visibility <- "Low_box_DB_Current_Time_1"
      HorizontalMovement <- "Low_box_DB_Current_Time_1"
   GraphicView "Graphic view_10" at 283,301 size 64x38; Picture "Graphic_25"
      Visibility <- "Low_box_DB_Current_Time_2"
      HorizontalMovement <- "Low_box_DB_Current_Time_2"
   GraphicView "Graphic view_12" at 283,301 size 64x38; Picture "Graphic_25"
      Visibility <- "Low_box_DB_Current_Time_3"
      HorizontalMovement <- "Low_box_DB_Current_Time_3"
   GraphicView "Graphic view_18" at 283,301 size 64x38; Picture "Graphic_25"
      Visibility <- "Low_box_DB_Current_Time_4"
      HorizontalMovement <- "Low_box_DB_Current_Time_4"
   GraphicView "Graphic view_19" at 283,301 size 64x38; Picture "Graphic_25"
      Visibility <- "Low_box_DB_Current_Time_5"
      HorizontalMovement <- "Low_box_DB_Current_Time_5"
   Circle "Circle_3" at 150,311 size 39x39
      Appearance <- "Run"
   GraphicView "Graphic view_21" at 796,240 size 71x78; Picture "Graphic_44"
   Circle "Circle_4" at 819,203 size 28x28
      Appearance <- "Piston_High"
   GraphicView "Graphic view_22" at 780,274 size 57x56; Picture "Graphic_55"
      Visibility <- "Piston_High"
   GraphicView "Graphic view_23" at 760,254 size 64x85; Picture "Graphic_25"
      DiagonalMovement <- "Control_Piston_High_DB_Multiple_boxes_Current_Time_1"
      Visibility <- "Control_Piston_High_DB_Multiple_boxes_Current_Time_1"
   Circle "Circle_5" at 692,59 size 36x36
      Appearance <- "Sensor_High"
   Button "Button_5" at 140,46 size 85x50; TextOff 'Low'
      on Release: ResetBit("Low")
      on Press: SetBit("Low")
   GraphicView "Graphic view_24" at 283,254 size 64x85; Picture "Graphic_25"
      Visibility <- "Control_Piston_High_DB_Multiple_boxes_Current_Time_1"
      HorizontalMovement <- "Control_Piston_High_DB_Multiple_boxes_Current_Time_1"
   GraphicView "Graphic view_20" at 283,254 size 64x85; Picture "Graphic_25"
      Visibility <- "Control_Piston_High_DB_Multiple_boxes_Current_Time_2"
      HorizontalMovement <- "Control_Piston_High_DB_Multiple_boxes_Current_Time_2"
   GraphicView "Graphic view_25" at 760,254 size 64x85; Picture "Graphic_25"
      DiagonalMovement <- "Control_Piston_High_DB_Multiple_boxes_Current_Time_3"
      Visibility <- "Control_Piston_High_DB_Multiple_boxes_Current_Time_3"
   GraphicView "Graphic view_27" at 283,254 size 64x85; Picture "Graphic_25"
      Visibility <- "Control_Piston_High_DB_Multiple_boxes_Current_Time_3"
      HorizontalMovement <- "Control_Piston_High_DB_Multiple_boxes_Current_Time_3"
   GraphicView "Graphic view_28" at 760,254 size 64x85; Picture "Graphic_25"
      DiagonalMovement <- "Control_Piston_High_DB_Multiple_boxes_Current_Time_2"
      Visibility <- "Control_Piston_High_DB_Multiple_boxes_Current_Time_2"
   GraphicView "Graphic view_29" at 283,254 size 64x85; Picture "Graphic_25"
      Visibility <- "Control_Piston_High_DB_Multiple_boxes_Current_Time_4"
      HorizontalMovement <- "Control_Piston_High_DB_Multiple_boxes_Current_Time_4"
   GraphicView "Graphic view_30" at 283,254 size 64x85; Picture "Graphic_25"
      Visibility <- "Control_Piston_High_DB_Multiple_boxes_Current_Time_5"
      HorizontalMovement <- "Control_Piston_High_DB_Multiple_boxes_Current_Time_5"
   GraphicView "Graphic view_31" at 760,254 size 64x85; Picture "Graphic_25"
      Visibility <- "Control_Piston_High_DB_Multiple_boxes_Current_Time_4"
      DiagonalMovement <- "Control_Piston_High_DB_Multiple_boxes_Current_Time_4"
   GraphicView "Graphic view_32" at 760,254 size 64x85; Picture "Graphic_25"
      DiagonalMovement <- "Control_Piston_High_DB_Multiple_boxes_Current_Time_5"
      Visibility <- "Control_Piston_High_DB_Multiple_boxes_Current_Time_5"
   GraphicView "Graphic view_33" at 283,277 size 64x64; Picture "Graphic_25"
      Visibility <- "Control_Piston_Med_DB_Multiple_boxes_Current_Time_1"
      HorizontalMovement <- "Control_Piston_Med_DB_Multiple_boxes_Current_Time_1"
   GraphicView "Graphic view_34" at 283,277 size 64x64; Picture "Graphic_25"
      Visibility <- "Control_Piston_Med_DB_Multiple_boxes_Current_Time_2"
      HorizontalMovement <- "Control_Piston_Med_DB_Multiple_boxes_Current_Time_2"
   GraphicView "Graphic view_35" at 283,277 size 64x64; Picture "Graphic_25"
      Visibility <- "Control_Piston_Med_DB_Multiple_boxes_Current_Time_3"
      HorizontalMovement <- "Control_Piston_Med_DB_Multiple_boxes_Current_Time_3"
   GraphicView "Graphic view_36" at 283,277 size 64x64; Picture "Graphic_25"
      Visibility <- "Control_Piston_Med_DB_Multiple_boxes_Current_Time_4"
      HorizontalMovement <- "Control_Piston_Med_DB_Multiple_boxes_Current_Time_4"
   GraphicView "Graphic view_37" at 283,277 size 64x64; Picture "Graphic_25"
      Visibility <- "Control_Piston_Med_DB_Multiple_boxes_Current_Time_5"
      HorizontalMovement <- "Control_Piston_Med_DB_Multiple_boxes_Current_Time_5"
   Button "Button_6" at 140,110 size 85x50; TextOff 'Med'
      on Release: ResetBit("Medium")
      on Press: SetBit("Medium")
   IOField "I/O field_2" at 1023,74 size 62x36; FormatPattern 999
      ProcessValue <- "DB_Main_Number_of_med_boxes"
   IOField "I/O field_3" at 762,74 size 62x36; FormatPattern 999
      ProcessValue <- "DB_Main_Number_of_high_boxes"
   GraphicView "Graphic view_38" at 946,98 size 56x134; Picture "Graphic_18"
   Circle "Circle_6" at 957,52 size 36x36
      Appearance <- "Sensor_Medium"
   SymbolLibrary "Symbol library_1" at 160,509 size 195x120
   SymbolLibrary "Symbol library_2" at 445,509 size 195x120
   SymbolLibrary "Symbol library_3" at 856,375 size 300x131
*)